FUNCTION_BLOCK FB_Vacuum EXTENDS FB_Device
VAR_INPUT
	bGrip							: BOOL;
	Timeout							: TIME;
END_VAR
VAR_OUTPUT
	Vacuum_Ok						: BOOL;
	Blow_Ok							: BOOL;
END_VAR
VAR
	VacuumValve				AT %Q*	: BOOL;
	BlowValve				AT %Q*	: BOOL;
	VaccumSensor			AT %I*	: BOOL;
	tmrBlow							: TP;
END_VAR

//	If execute grip input then grip
	VacuumValve						:=	bGrip;
	BlowValve						:=	(NOT bGrip) AND VaccumSensor;

//	Assing valiue to function block status
	Vacuum_Ok							:= VaccumSensor AND NOT BlowValve;
	Blow_Ok								:= BlowValve AND NOT VacuumValve;

//	For setting alarms
	Alarm();

METHOD Alarm
//	Timer for set action executing timeout alarm
	ton_StepTimeout(		IN:=(VacuumValve AND (NOT VaccumSensor)) OR (BlowValve AND VaccumSensor),
							PT:=Timeout);

//	For no vacc sensor feedback alarm setting
	AlarmCodesHandling(sConcatCodes:=sAlarm,sCode:='EVACUDET01 ',sIDToAdd:=sDeviceID,bActive:=(VacuumValve AND ton_StepTimeout.Q));
//	For no release success alarm setting
	AlarmCodesHandling(sConcatCodes:=sAlarm,sCode:='EVACUDET02 ',sIDToAdd:=sDeviceID,bActive:=(BlowValve AND ton_StepTimeout.Q));
END_METHOD

METHOD Pick : bool
VAR_INPUT	
END_VAR
BlowValve:= FALSE;
VacuumValve:= TRUE;

//IF NOT VaccumSensor THEN
//	SetAlarm('Vacuum not reached!');
//ELSE
//	SetAlarm('');	
//END_IF

Pick := VaccumSensor;
END_METHOD

METHOD Release : bool
VAR_INPUT
	Blow			: BOOL 	:= FALSE;
	BlowPulse		: TIME	:= T#100MS;
END_VAR
VacuumValve:= FALSE;
tmrBlow(In:= TRUE, PT:= BlowPulse);

IF blow AND tmrBlow.Q THEN
	BlowValve:= TRUE;
ELSE
	BlowValve:= FALSE;		
END_IF



Release := NOT VaccumSensor AND tmrBlow.Q;
END_METHOD

END_FUNCTION_BLOCK

(* stored: Version 1.1.0.1, ProductVersion 3.1.4024.12
   POU FB_Vacuum: Id {f9531b35-4007-4908-8918-76526d36fc74}, SpecialFunc None
   Method Alarm: Id {8de2fcf2-2e3b-4735-b382-f976ceab4d57}
   Method Pick: Id {7a8bb277-e95f-446d-a6b9-288a0c9e0a5c}
   Method Release: Id {fecf298a-d878-4a03-bda7-5624c8bf16fd} *)
